Staubli VAL3: writeStrValue.pgx

public program writeStrValue(num x_nCamID (dimensions=1), string x_sCellNumber (dimensions=1), string x_sMsg (dimensions=1), bool& x_bError[] (dimensions=1))
  local string l_sCell
  local bool l_bIsOk
begin
  //-----------------------------------------------------------------------
  //Header begin
  //Description of program
  //  Sets an edit box control contained in a cell (x_sCellNumber) to a
  //  specified string (x_sMsg)
  //  The target cell of the writing operation in the Cognex spreadsheet must
  //  be of the EditString type.
  //
  //Input parameters
  //  num x_nCamID :
  //    role : camera's ID
  //  string x_sCellNumber :
  //    role : The column letter and the row number of the cell value to get.
  //    possible values : - column letter : (A to Z)
  //                      - row number : (000 to 399)
  //  string x_sMsg :
  //    role : string to writing in the cell
  //
  //Output parameters
  //  bool x_bError :
  //    role : returns false if operation suceeded and true otherwise
  //
  //Examples
  //  call writeStrValue(nCamID,"C6","Example Staubli",l_bError)
  //
  //History
  //  Creation : 19-05-08 - f.Rob
  //Header end
  //-----------------------------------------------------------------------

  x_bError=true
  call checkCellFormat(x_nCamID,x_sCellNumber,l_bIsOk)
  if l_bIsOk
    nProgram[x_nCamID]=11
    call sendCommand(x_nCamID,"SS"+x_sCellNumber+x_sMsg,x_bError)
  endIf
end
